(* PLC project Generated.project, CODESYS CODESYS V3.5 SP19 Patch 1 *)
(* stored: creationDateTime 2026-08-28T11:10:17.737492, modificationDateTime 2026-08-28T11:10:17.737492 *)

(* ═══════════════════════════════════════════════════════════════ ST_DredgingAssistCfg — Réglages persistants assistants prélèvement 📄 Doc : DOC/AF/AF_Partie-04_Mode_SemiAuto_Sequenceur_v2.3.md §3ter ═══════════════════════════════════════════════════════════════ *)
TYPE ST_DredgingAssistCfg : STRUCT
  DiveStartMin_M : REAL := 1;  (* Position mini M1/M2 avant plongée *)
  ImmersionUpper_M : REAL := 0.5;  (* Borne haute fenêtre front immersion *)
  ImmersionLower_M : REAL := -0.5;  (* Borne basse fenêtre front immersion *)
  ExtractionControlDistance_M : REAL := 2;  (* Remontée palier 1 avant accélération *)
  TglEnableDiveSearch : BOOL := FALSE;  (* Mode assistance plongée mémorisé *)
  TglEnableExtractionSequence : BOOL := FALSE;  (* Mode assistance extraction mémorisé *)
  TglEnableDumpAtTremie : BOOL := FALSE;  (* Mode assistance vidage trémie mémorisé *)
  Initialized : BOOL := FALSE;  (* Pont persistance/IHM initialisé *)
END_STRUCT;
END_TYPE
